TYPE ST_ConfigFeatures :
STRUCT
    ExportCurrentConfig : BOOL;
END_STRUCT
END_TYPE

(* stored: Version 1.1.0.1, ProductVersion 3.1.4024.12
   DUT ST_ConfigFeatures: Id {4eced73f-d97b-45f7-bece-6539fadfd530} *)
